TYPE DUT :
UNION
END_UNION
END_TYPE

(* stored: Version 1.1.0.1, ProductVersion 3.1.4024.14
   DUT DUT: Id {7195751e-d8a1-4708-8748-f03988e8de87} *)
